// Mitsubishi GX Works2 project: 액츄에이터제어 평가   PLC: Q02/Q02H

PROGRAM MAIN
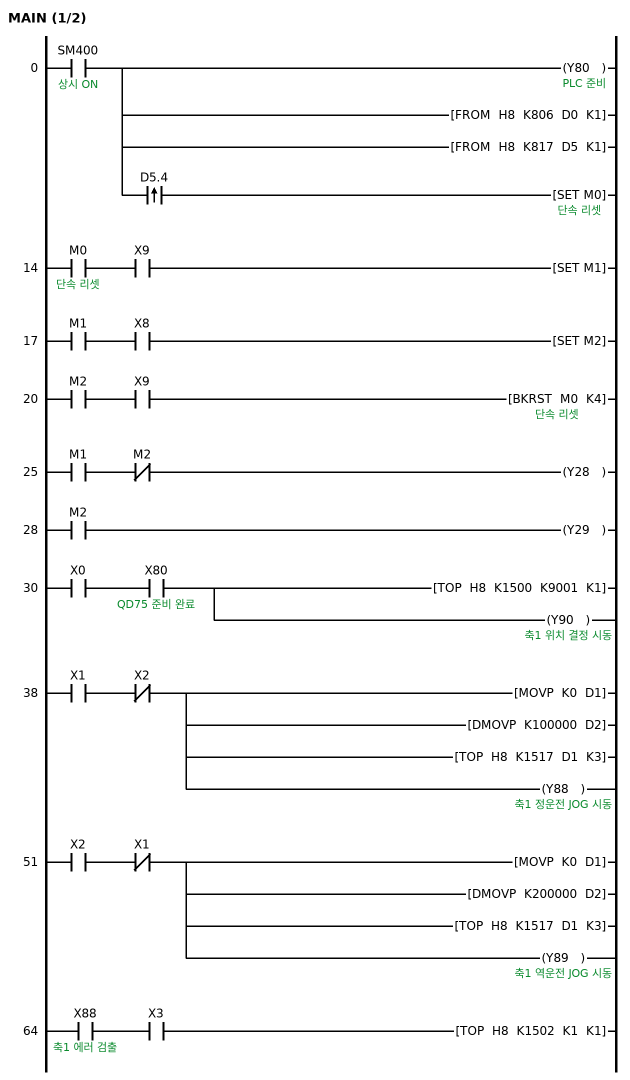
0     LD      SM400  ; 상시 ON
      OUT     Y80  ; PLC 준비
      FROM    H8 K806 D0 K1
      FROM    H8 K817 D5 K1
      ANDP    D5.4
      SET     M0  ; 단속 리셋
14    LD      M0  ; 단속 리셋
      AND     X9
      SET     M1
17    LD      M1
      AND     X8
      SET     M2
20    LD      M2
      AND     X9
      BKRST   M0 K4
25    LD      M1
      ANI     M2
      OUT     Y28
28    LD      M2
      OUT     Y29
30    LD      X0
      AND     X80  ; QD75 준비 완료
      TOP     H8 K1500 K9001 K1
      OUT     Y90  ; 축1 위치 결정 시동
38    LD      X1
      ANI     X2
      MOVP    K0 D1
      DMOVP   K100000 D2
      TOP     H8 K1517 D1 K3
      OUT     Y88  ; 축1 정운전 JOG 시동
51    LD      X2
      ANI     X1
      MOVP    K0 D1
      DMOVP   K200000 D2
      TOP     H8 K1517 D1 K3
      OUT     Y89  ; 축1 역운전 JOG 시동
64    LD      X88  ; 축1 에러 검출
      AND     X3
      TOP     H8 K1502 K1 K1
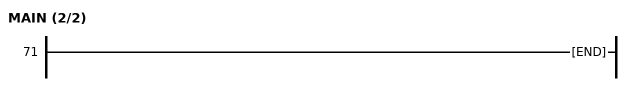
71    END
END_PROGRAM

// device comments not shown above
X81  ; 동기용 플래그
X84  ; 축1 M 코드 ON
X85  ; 축2 M 코드 ON
X89  ; 축2 에러 검출
X8C  ; 축1 BUSY
X8D  ; 축2 BUSY
X90  ; 축1 시동 완료
X91  ; 축2 시동 완료
X94  ; 축1 위치 결정 완료
X95  ; 축2 위치 결정 완료
Y84  ; 축1 축 정지
Y85  ; 축2 축 정지
Y8A  ; 축2 정운전 JOG 시동
Y8B  ; 축2 역운전 JOG 시동
Y91  ; 축2 위치 결정 시동
Y94  ; 축1 실행 금지 플래그
Y95  ; 축2 실행 금지 플래그
M11  ; 공_전
M12  ; 공_후
M13  ; 가공모터 회전
M14  ; 드_하
M15  ; 드_상
M16  ; 가공모터 정지
M17  ; 송_전
M18  ; 송_후
M19  ; 컨베이어 구동
M20  ; 동작끝
M21  ; 비금속
M22  ; 스_하
M23  ; 컨베이어 정지
M24  ; 서보 리프트 하강
M25  ; 흡착패드 동작
M26  ; 서보 리프트 이동
M27  ; 흡_전
M28  ; 흡착패드 정지
M29  ; 흡_후
M30  ; 원점 복귀
M31  ; 스토퍼실린더 상승
M32  ; 종료리셋
M50  ; 금속
M100  ; 연속동작
M101  ; 연속동작 종료
M200  ; 연속동작 금속
M300  ; 연속동작 비금속
M800  ; 연속리셋
M1000  ; 연속시작
M1500  ; 연속시작
M1900  ; 연속리셋
T1  ; 2초 지연
T2  ; 8초 동작
T3  ; 2초 지연
T100  ; 연속리셋타이머
D100  ; 연속동작
D200  ; 연속트리거
D300  ; 비금속개수
D310  ; 금속개수
